% RSLogix 500 project P5.RSS, saved by version 12.00.00.00 %
PROJECT "UNTITLED"    % processor: Bul.1763 MicroLogix 1100 Series B %

PROGRAM FILES
  LAD 2   6 rungs

DATA FILES
  O0 OUTPUT  4 elements
  I1 INPUT  6 elements
  S2 STATUS  66 elements
  B3 BINARY  1 elements
  T4 TIMER  3 elements
  C5 COUNTER  1 elements
  R6 CONTROL  1 elements
  N7 INTEGER  1 elements
  F8 FLOAT  3 elements

LADDER 2
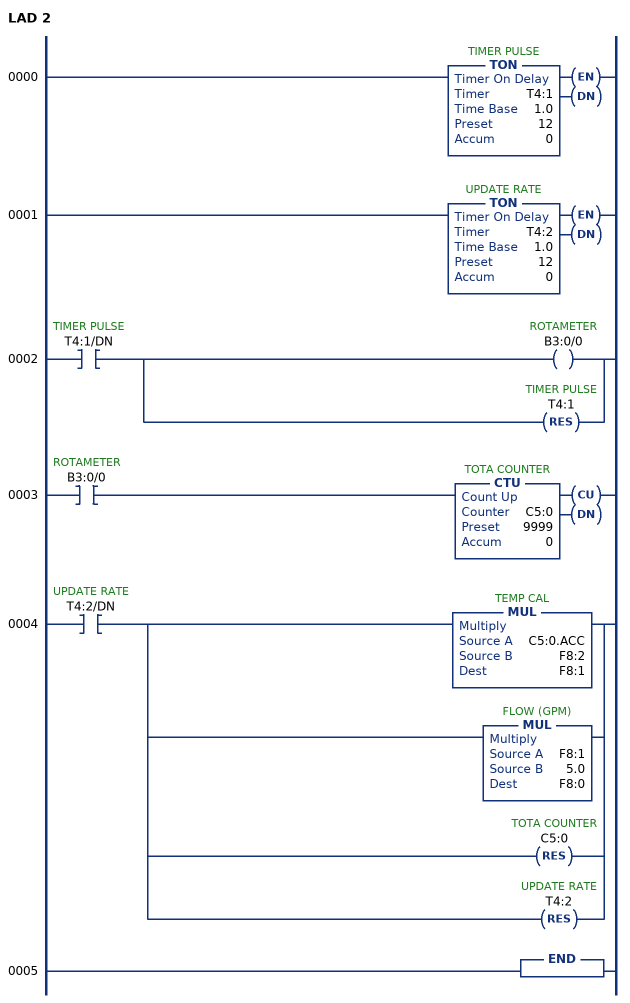
% Rung: 0 %
SOR TON T4:1 1.0 12 0 EOR
%   T4:1  "TIMER PULSE" %
% Rung: 1 %
SOR TON T4:2 1.0 12 0 EOR
%   T4:2  "UPDATE RATE" %
% Rung: 2 %
SOR XIC T4:1/DN BST OTE B3:0/0 NXB RES T4:1 BND EOR
%   T4:1/DN  "TIMER PULSE" %
%   B3:0/0  "ROTAMETER" %
%   T4:1  "TIMER PULSE" %
% Rung: 3 %
SOR XIC B3:0/0 CTU C5:0 9999 0 EOR
%   B3:0/0  "ROTAMETER" %
%   C5:0  "TOTA COUNTER" %
% Rung: 4 %
SOR XIC T4:2/DN BST MUL C5:0.ACC F8:2 F8:1 NXB MUL F8:1 5.0 F8:0 NXB RES C5:0 NXB RES T4:2 BND EOR
%   T4:2  "UPDATE RATE" %
%   C5:0  "TOTA COUNTER" %
%   F8:2  "k FACTOR" %
%   F8:1  "TEMP CAL" %
%   F8:0  "FLOW (GPM)" %
% Rung: 5 %
SOR END EOR

OTHER DOCUMENTED ADDRESSES
  B3:0/1  "UPDATE RESET"
  N7:0  "PULSE COUNTED"
  T4:0  "SYSTEM TIMER"

DATA TABLE (non-zero values as saved)
DATA T4
% .PRE .ACC %
% T4:0 % 60 0
% T4:1 % 12 0
% T4:2 % 12 0
DATA C5
% .PRE .ACC %
% C5:0 % 9999 0
